(* Logix 5000 project; controller Good_Foods_96985_10252022_1208 vendor 1 type 14 code 151 rev 32.15; software revision 32.04; part 4 of 4 *)
(* tags used below, declared in another part *)
   Auto_Reset_Timer : TIMER;
   Auto_Reset_Timer2 : TIMER;
   bActive_Cleanout_Mode : BOOL;
   bAll_Doors_OK : BOOL;
   bAll_EStops_OK : BOOL;
   bAuto_Clear_Faults : BOOL;
   bAuto_Disable_Servos : BOOL;
   bAuto_Enable_Servos : BOOL;
   bAuto_Enable_VFDs : BOOL;
   bAuto_Reset_Latch : BOOL;
   bAuto_Reset_Servos : BOOL;
   bBatch_Cmplt : BOOL;
   bHMI_IND_Alarm_Active : BOOL;
   bHMI_IND_Servos_Enable : BOOL;
   bHMI_PB_Fault_Reset : BOOL;
   bHMI_PB_Jog_Infeed_Conveyors : BOOL;
   bHMI_PB_JogFwd_Left_Denester : BOOL;
   bHMI_PB_JogFwd_Right_Denester : BOOL;
   bHMI_PB_JogRev_Left_Denester : BOOL;
   bHMI_PB_JogRev_Right_Denester : BOOL;
   bHMI_PB_Left_Denester_Enabled : BOOL;
   bHMI_PB_Right_Denester_Enabled : BOOL;
   bLeft_System_Not_Running : BOOL;
   bLeftConvBacklog_OK : BOOL;
   bLeftDropBacklog_OK : BOOL;
   bLeftPrimeBacklog_OK : BOOL;
   bMachine_Startup_Delay : BOOL;
   bRight_System_Not_Running : BOOL;
   bRightConvBacklog_OK : BOOL;
   bRightDropBacklog_OK : BOOL;
   bRightPrimeBacklog_OK : BOOL;
   bSafety_OK : BOOL;
   bSystem_Active : BOOL;
   bSystem_Alarm_Active : BOOL;
   bSystem_Conveyor_Run_Perm : BOOL;
   bSystem_Needs_To_Be_Homed : BOOL;
   bSystem_VFDStop_CMPLT : BOOL;
   dAlarms : DINT[8];
   DI_Estop_Autoloader_Pressed : BOOL;
   DI_Estop_HMI_Pressed : BOOL;
   DI_Estop_NonOpSide_Pressed : BOOL;
   DI_PB_Autoloader_Start : BOOL;
   DI_PB_Hmi_Jog : BOOL;
   DI_PRX_Left_DropGate_EXT : BOOL;
   DI_PRX_Left_DropGate_RET : BOOL;
   DI_PRX_Left_Shuttle_RET : BOOL;
   DI_PRX_Right_DropGate_EXT : BOOL;
   DI_PRX_Right_DropGate_RET : BOOL;
   DI_PRX_Right_Shuttle_RET : BOOL;
   DI_PS_Air_Supply_OK : BOOL;
   DI_Safety_Relay_OK : BOOL;
   DI_SS_Left_NonOp_Door_Open : BOOL;
   DI_SS_Left_Op_Door_Open : BOOL;
   DI_SS_Right_NonOp_Door_Open : BOOL;
   DI_SS_Right_Op_Door_Open : BOOL;
   dLeft_Shuttle_Seq_CMD : DINT;
   dRight_Shuttle_Seq_CMD : DINT;
   intStatus_Message : INT;
   Left_Container_Jam_Timer : TIMER;
   Left_Denester : AXIS_CIP_DRIVE;
   Left_Rev_Count : INT;
   Master_Encoder : AXIS_CIP_DRIVE;
   ONS : DINT[16];
   rConv_Speed : REAL;
   rConv_Speed_Hz : DINT;
   rHMI_Infeed_Conv_Multiplier : REAL;
   rHMI_Machine_Speed : REAL;
   Right_Container_Jam_Timer : TIMER;
   Right_Denester : AXIS_CIP_DRIVE;
   Right_Rev_Count : INT;
   Timer_AirPressure : TIMER;
   tLeftDropGateContTimeOut : TIMER;
   tLeftDropGateExtTimeOut : TIMER;
   tLeftDropGateOpenTimeOut : TIMER;
   tLeftShuttleContPresTimeOut : TIMER;
   tloadconvpress : TIMER;
   tRightDropGateContTimeOut : TIMER;
   tRightDropGateExtTimeOut : TIMER;
   tRightDropGateOpenTimeOut : TIMER;
   tRightShuttleContPresTimeOut : TIMER;
(* MainProgram, continued *)

ROUTINE _30_VFDs   (* ladder *)
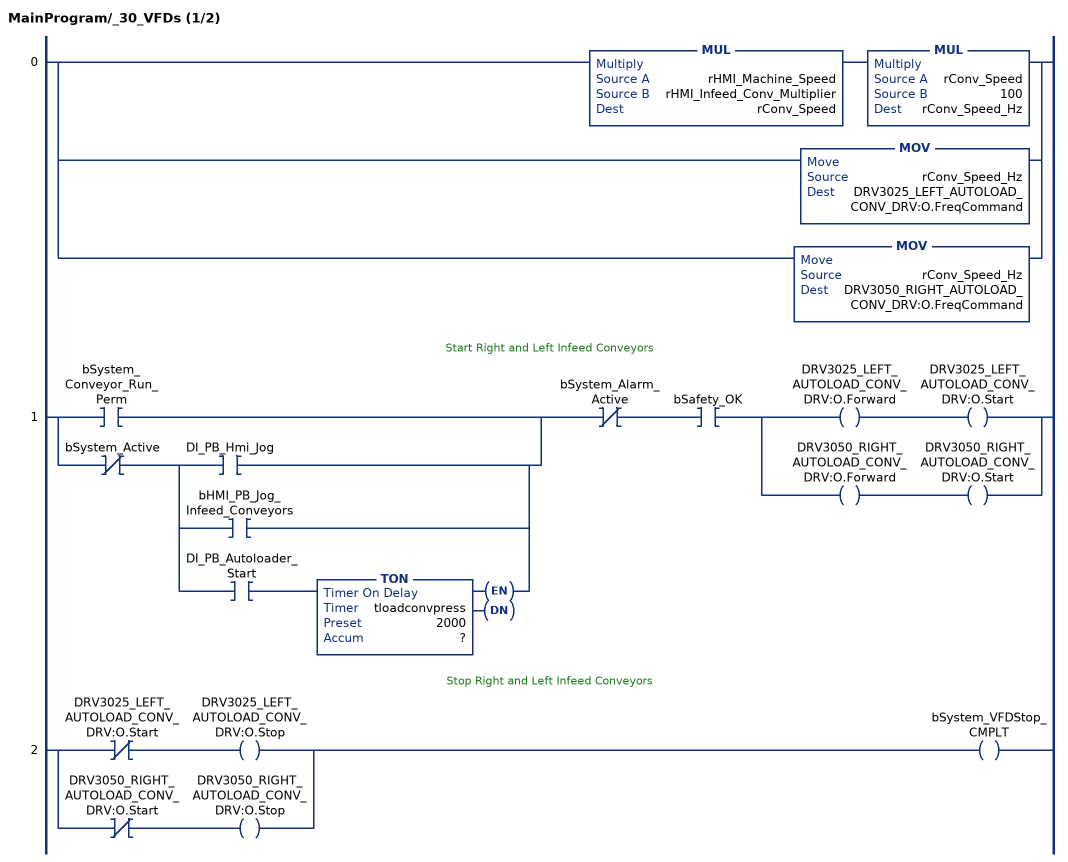
   0: [MUL(rHMI_Machine_Speed,rHMI_Infeed_Conv_Multiplier,rConv_Speed) MUL(rConv_Speed,100,rConv_Speed_Hz) ,MOV(rConv_Speed_Hz,DRV3025_LEFT_AUTOLOAD_CONV_DRV:O.FreqCommand) ,MOV(rConv_Speed_Hz,DRV3050_RIGHT_AUTOLOAD_CONV_DRV:O.FreqCommand) ];
   // Start Right and Left Infeed Conveyors
   1: [XIC(bSystem_Conveyor_Run_Perm) ,XIO(bSystem_Active) [XIC(DI_PB_Hmi_Jog) ,XIC(bHMI_PB_Jog_Infeed_Conveyors) ,XIC(DI_PB_Autoloader_Start) TON(tloadconvpress,?,?) ] ]XIO(bSystem_Alarm_Active)XIC(bSafety_OK)[OTE(DRV3025_LEFT_AUTOLOAD_CONV_DRV:O.Forward) OTE(DRV3025_LEFT_AUTOLOAD_CONV_DRV:O.Start) ,OTE(DRV3050_RIGHT_AUTOLOAD_CONV_DRV:O.Forward) OTE(DRV3050_RIGHT_AUTOLOAD_CONV_DRV:O.Start) ];
   // Stop Right and Left Infeed Conveyors
   2: [XIO(DRV3025_LEFT_AUTOLOAD_CONV_DRV:O.Start) OTE(DRV3025_LEFT_AUTOLOAD_CONV_DRV:O.Stop) ,XIO(DRV3050_RIGHT_AUTOLOAD_CONV_DRV:O.Start) OTE(DRV3050_RIGHT_AUTOLOAD_CONV_DRV:O.Stop) ]OTE(bSystem_VFDStop_CMPLT);
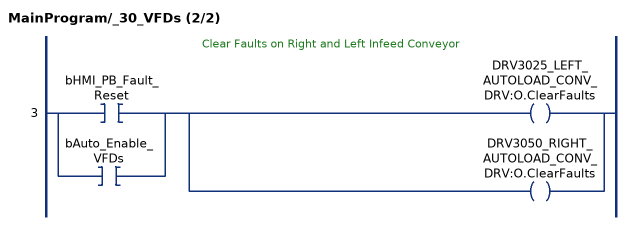
   // Clear Faults on Right and Left Infeed Conveyor
   3: [XIC(bHMI_PB_Fault_Reset) ,XIC(bAuto_Enable_VFDs) ][OTE(DRV3025_LEFT_AUTOLOAD_CONV_DRV:O.ClearFaults) ,OTE(DRV3050_RIGHT_AUTOLOAD_CONV_DRV:O.ClearFaults) ];
END_ROUTINE

ROUTINE _90_Status_Messages   (* ladder *)
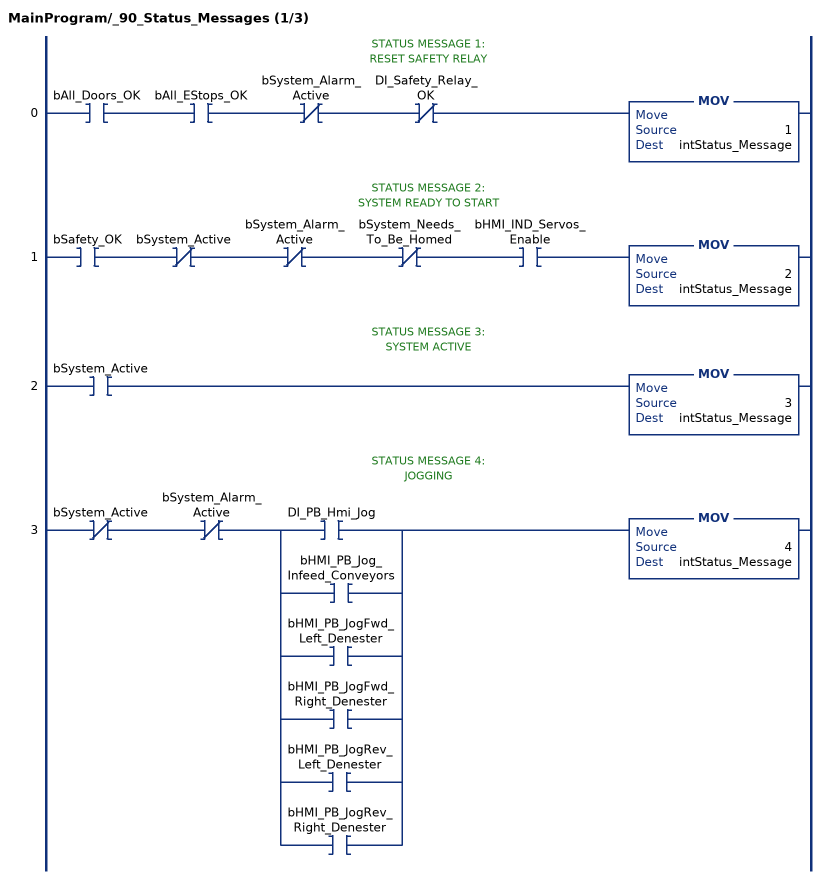
   // STATUS MESSAGE 1:
   // RESET SAFETY RELAY
   0: XIC(bAll_Doors_OK)XIC(bAll_EStops_OK)XIO(bSystem_Alarm_Active)XIO(DI_Safety_Relay_OK)MOV(1,intStatus_Message);
   // STATUS MESSAGE 2:
   // SYSTEM READY TO START
   1: XIC(bSafety_OK)XIO(bSystem_Active)XIO(bSystem_Alarm_Active)XIO(bSystem_Needs_To_Be_Homed)XIC(bHMI_IND_Servos_Enable)MOV(2,intStatus_Message);
   // STATUS MESSAGE 3:
   // SYSTEM ACTIVE
   2: XIC(bSystem_Active)MOV(3,intStatus_Message);
   // STATUS MESSAGE 4:
   // JOGGING
   3: XIO(bSystem_Active)XIO(bSystem_Alarm_Active)[XIC(DI_PB_Hmi_Jog) ,XIC(bHMI_PB_Jog_Infeed_Conveyors) ,XIC(bHMI_PB_JogFwd_Left_Denester) ,XIC(bHMI_PB_JogFwd_Right_Denester) ,XIC(bHMI_PB_JogRev_Left_Denester) ,XIC(bHMI_PB_JogRev_Right_Denester) ]MOV(4,intStatus_Message);
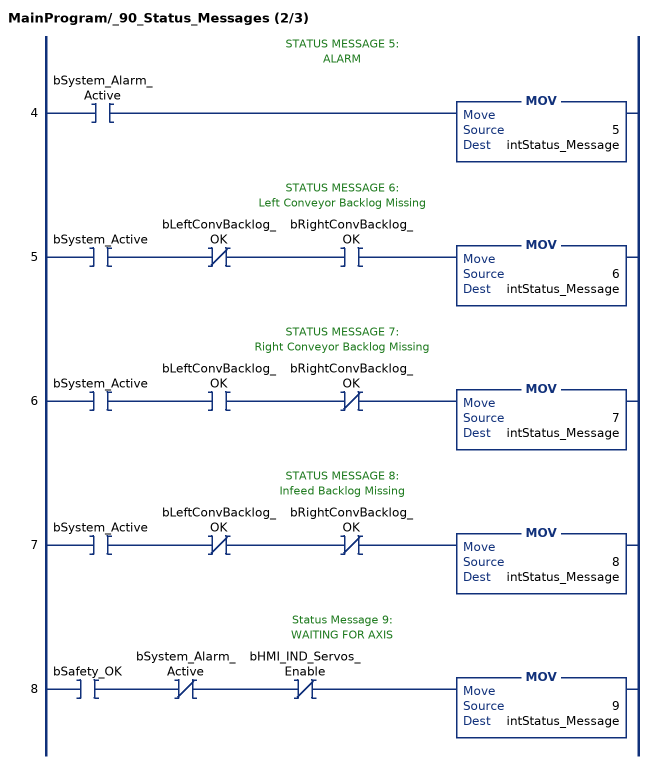
   // STATUS MESSAGE 5:
   // ALARM
   4: XIC(bSystem_Alarm_Active)MOV(5,intStatus_Message);
   // STATUS MESSAGE 6:
   // Left Conveyor Backlog Missing
   5: XIC(bSystem_Active)XIO(bLeftConvBacklog_OK)XIC(bRightConvBacklog_OK)MOV(6,intStatus_Message);
   // STATUS MESSAGE 7:
   // Right Conveyor Backlog Missing
   6: XIC(bSystem_Active)XIC(bLeftConvBacklog_OK)XIO(bRightConvBacklog_OK)MOV(7,intStatus_Message);
   // STATUS MESSAGE 8:
   // Infeed Backlog Missing
   7: XIC(bSystem_Active)XIO(bLeftConvBacklog_OK)XIO(bRightConvBacklog_OK)MOV(8,intStatus_Message);
   // Status Message 9:
   // WAITING FOR AXIS
   8: XIC(bSafety_OK)XIO(bSystem_Alarm_Active)XIO(bHMI_IND_Servos_Enable)MOV(9,intStatus_Message);
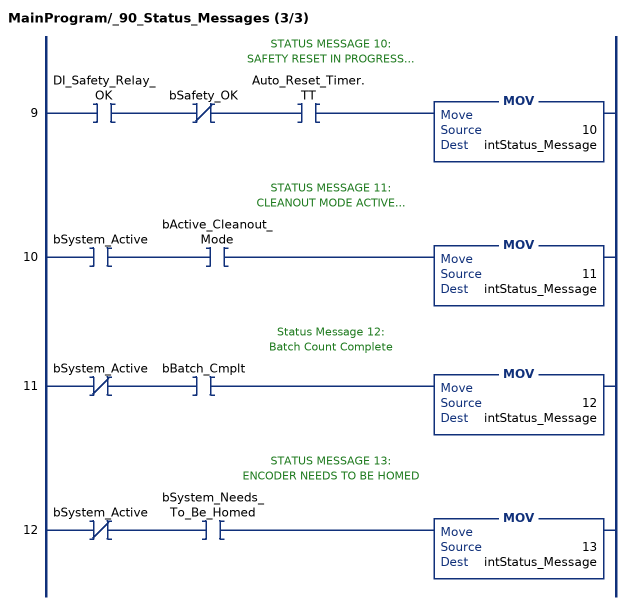
   // STATUS MESSAGE 10:
   // SAFETY RESET IN PROGRESS...
   9: XIC(DI_Safety_Relay_OK)XIO(bSafety_OK)XIC(Auto_Reset_Timer.TT)MOV(10,intStatus_Message);
   // STATUS MESSAGE 11:
   // CLEANOUT MODE ACTIVE...
   10: XIC(bSystem_Active)XIC(bActive_Cleanout_Mode)MOV(11,intStatus_Message);
   // Status Message 12:
   // Batch Count Complete
   11: XIO(bSystem_Active)XIC(bBatch_Cmplt)MOV(12,intStatus_Message);
   // STATUS MESSAGE 13:
   // ENCODER NEEDS TO BE HOMED
   12: XIO(bSystem_Active)XIC(bSystem_Needs_To_Be_Homed)MOV(13,intStatus_Message);
END_ROUTINE

ROUTINE _99_Alarms   (* ladder *)
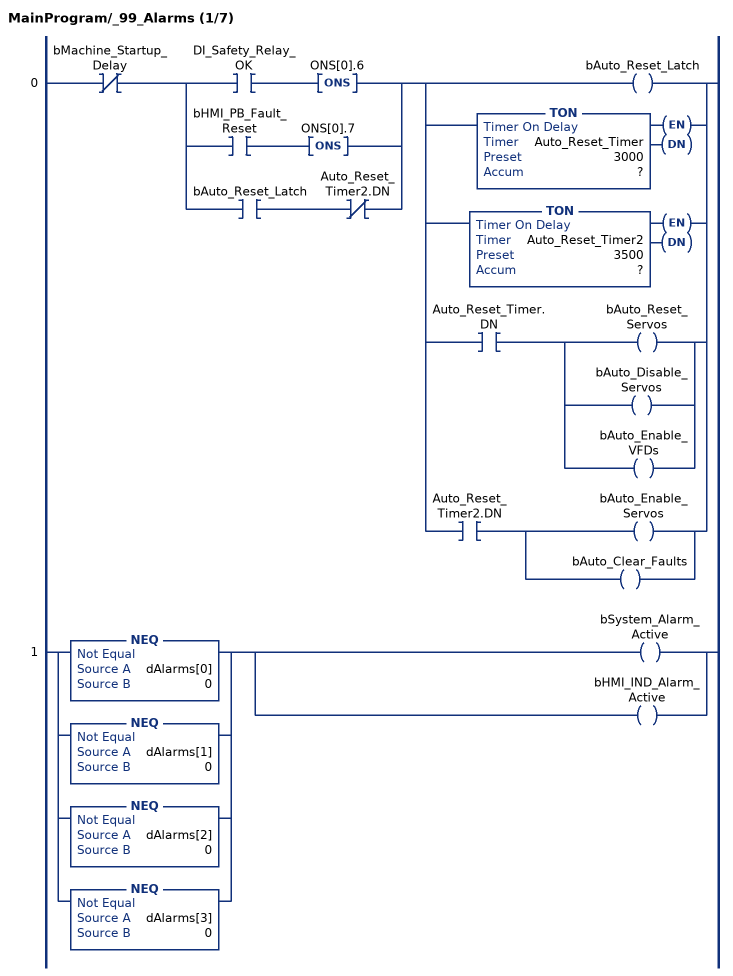
   0: XIO(bMachine_Startup_Delay)[XIC(DI_Safety_Relay_OK) ONS(ONS[0].6) ,XIC(bHMI_PB_Fault_Reset) ONS(ONS[0].7) ,XIC(bAuto_Reset_Latch) XIO(Auto_Reset_Timer2.DN) ][OTE(bAuto_Reset_Latch) ,TON(Auto_Reset_Timer,?,?) ,TON(Auto_Reset_Timer2,?,?) ,XIC(Auto_Reset_Timer.DN) [OTE(bAuto_Reset_Servos) ,OTE(bAuto_Disable_Servos) ,OTE(bAuto_Enable_VFDs) ] ,XIC(Auto_Reset_Timer2.DN) [OTE(bAuto_Enable_Servos) ,OTE(bAuto_Clear_Faults) ] ];
   1: [NEQ(dAlarms[0],0) ,NEQ(dAlarms[1],0) ,NEQ(dAlarms[2],0) ,NEQ(dAlarms[3],0) ][OTE(bSystem_Alarm_Active) ,OTE(bHMI_IND_Alarm_Active) ];
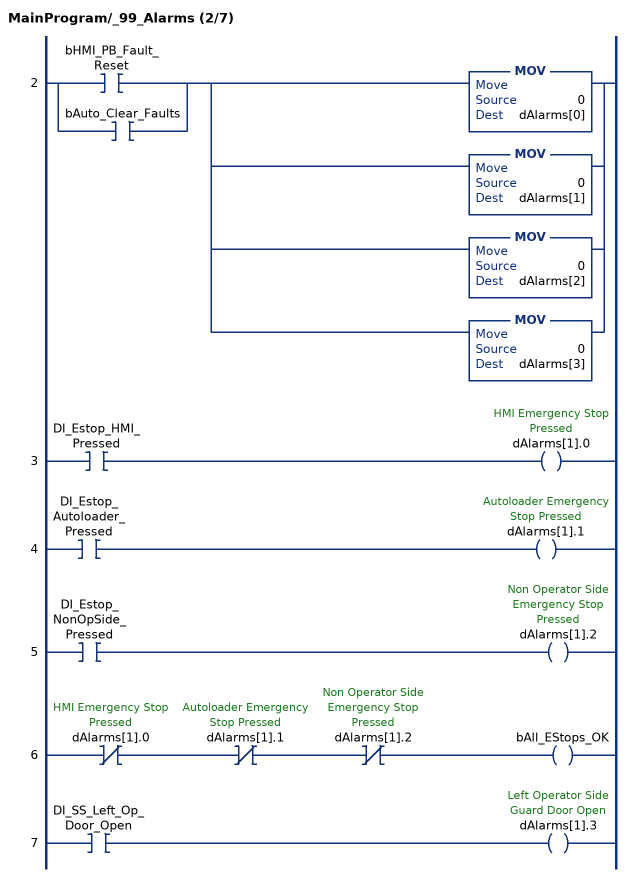
   2: [XIC(bHMI_PB_Fault_Reset) ,XIC(bAuto_Clear_Faults) ][MOV(0,dAlarms[0]) ,MOV(0,dAlarms[1]) ,MOV(0,dAlarms[2]) ,MOV(0,dAlarms[3]) ];
   3: XIC(DI_Estop_HMI_Pressed)OTE(dAlarms[1].0);
   4: XIC(DI_Estop_Autoloader_Pressed)OTE(dAlarms[1].1);
   5: XIC(DI_Estop_NonOpSide_Pressed)OTE(dAlarms[1].2);
   6: XIO(dAlarms[1].0)XIO(dAlarms[1].1)XIO(dAlarms[1].2)OTE(bAll_EStops_OK);
   7: XIC(DI_SS_Left_Op_Door_Open)OTE(dAlarms[1].3);
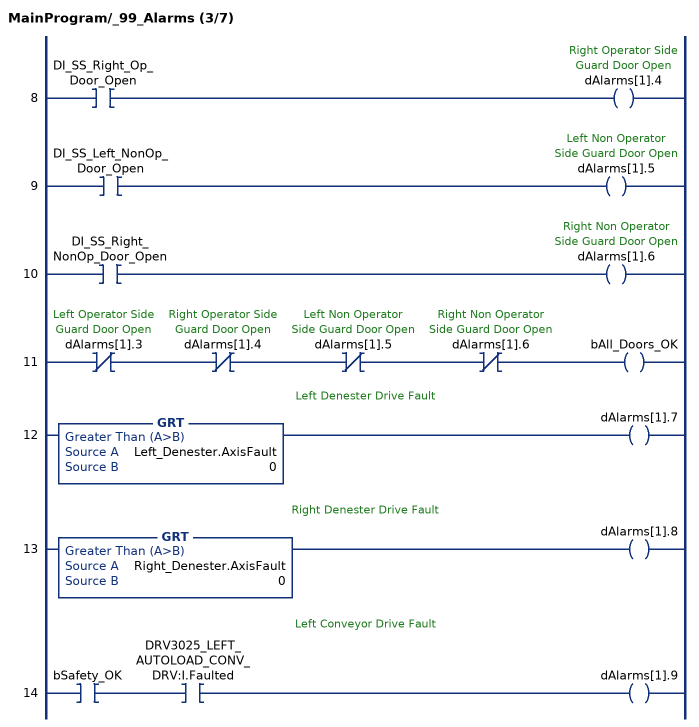
   8: XIC(DI_SS_Right_Op_Door_Open)OTE(dAlarms[1].4);
   9: XIC(DI_SS_Left_NonOp_Door_Open)OTE(dAlarms[1].5);
   10: XIC(DI_SS_Right_NonOp_Door_Open)OTE(dAlarms[1].6);
   11: XIO(dAlarms[1].3)XIO(dAlarms[1].4)XIO(dAlarms[1].5)XIO(dAlarms[1].6)OTE(bAll_Doors_OK);
   // Left Denester Drive Fault
   12: GRT(Left_Denester.AxisFault,0)OTE(dAlarms[1].7);
   // Right Denester Drive Fault
   13: GRT(Right_Denester.AxisFault,0)OTE(dAlarms[1].8);
   // Left Conveyor Drive Fault
   14: XIC(bSafety_OK)XIC(DRV3025_LEFT_AUTOLOAD_CONV_DRV:I.Faulted)OTE(dAlarms[1].9);
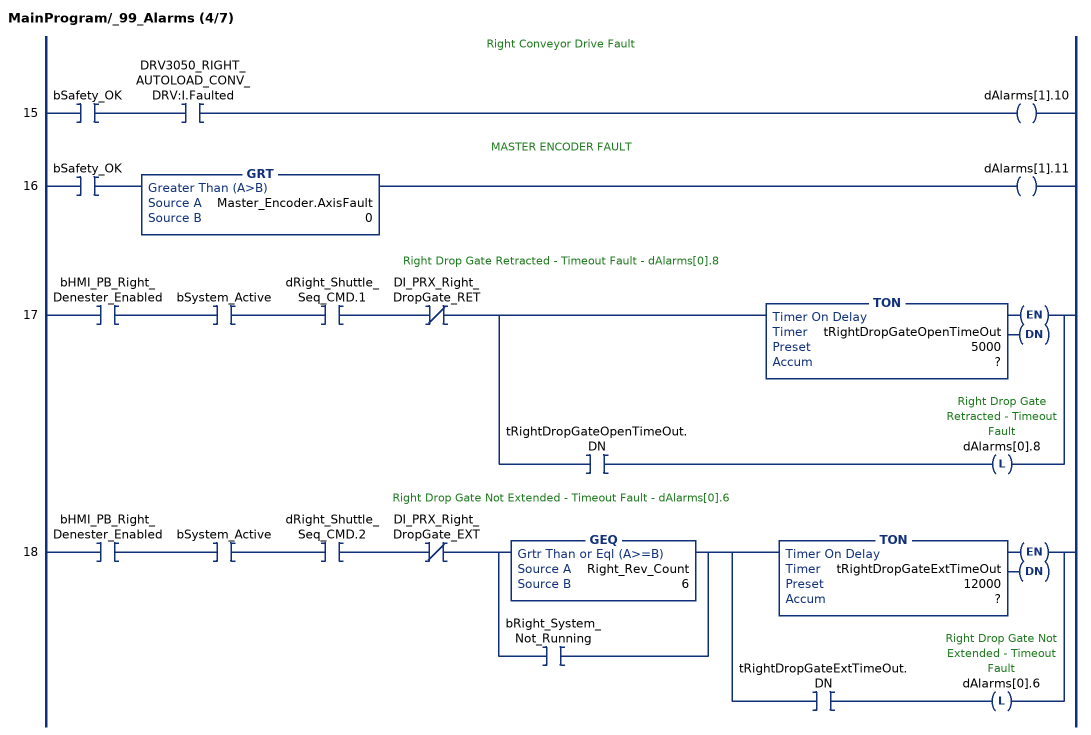
   // Right Conveyor Drive Fault
   15: XIC(bSafety_OK)XIC(DRV3050_RIGHT_AUTOLOAD_CONV_DRV:I.Faulted)OTE(dAlarms[1].10);
   // MASTER ENCODER FAULT
   16: XIC(bSafety_OK)GRT(Master_Encoder.AxisFault,0)OTE(dAlarms[1].11);
   // Right Drop Gate Retracted - Timeout Fault - dAlarms[0].8
   17: XIC(bHMI_PB_Right_Denester_Enabled)XIC(bSystem_Active)XIC(dRight_Shuttle_Seq_CMD.1)XIO(DI_PRX_Right_DropGate_RET)[TON(tRightDropGateOpenTimeOut,?,?) ,XIC(tRightDropGateOpenTimeOut.DN) OTL(dAlarms[0].8) ];
   // Right Drop Gate Not Extended - Timeout Fault - dAlarms[0].6
   18: XIC(bHMI_PB_Right_Denester_Enabled)XIC(bSystem_Active)XIC(dRight_Shuttle_Seq_CMD.2)XIO(DI_PRX_Right_DropGate_EXT)[GEQ(Right_Rev_Count,6) ,XIC(bRight_System_Not_Running) ][TON(tRightDropGateExtTimeOut,?,?) ,XIC(tRightDropGateExtTimeOut.DN) OTL(dAlarms[0].6) ];
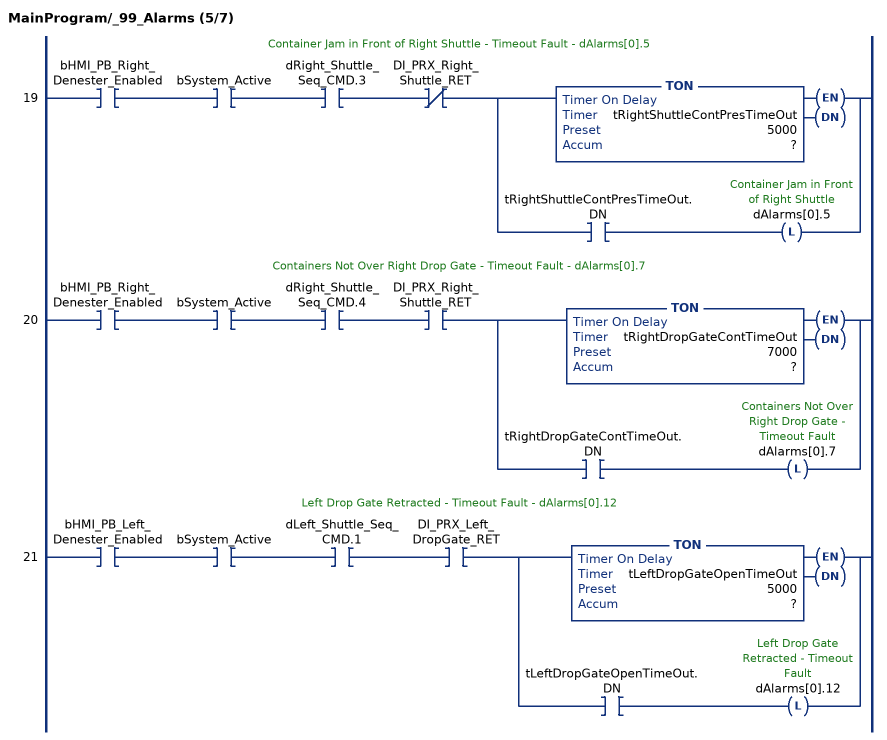
   // Container Jam in Front of Right Shuttle - Timeout Fault - dAlarms[0].5
   19: XIC(bHMI_PB_Right_Denester_Enabled)XIC(bSystem_Active)XIC(dRight_Shuttle_Seq_CMD.3)XIO(DI_PRX_Right_Shuttle_RET)[TON(tRightShuttleContPresTimeOut,?,?) ,XIC(tRightShuttleContPresTimeOut.DN) OTL(dAlarms[0].5) ];
   // Containers Not Over Right Drop Gate - Timeout Fault - dAlarms[0].7
   20: XIC(bHMI_PB_Right_Denester_Enabled)XIC(bSystem_Active)XIC(dRight_Shuttle_Seq_CMD.4)XIC(DI_PRX_Right_Shuttle_RET)[TON(tRightDropGateContTimeOut,?,?) ,XIC(tRightDropGateContTimeOut.DN) OTL(dAlarms[0].7) ];
   // Left Drop Gate Retracted - Timeout Fault - dAlarms[0].12
   21: XIC(bHMI_PB_Left_Denester_Enabled)XIC(bSystem_Active)XIC(dLeft_Shuttle_Seq_CMD.1)XIC(DI_PRX_Left_DropGate_RET)[TON(tLeftDropGateOpenTimeOut,?,?) ,XIC(tLeftDropGateOpenTimeOut.DN) OTL(dAlarms[0].12) ];
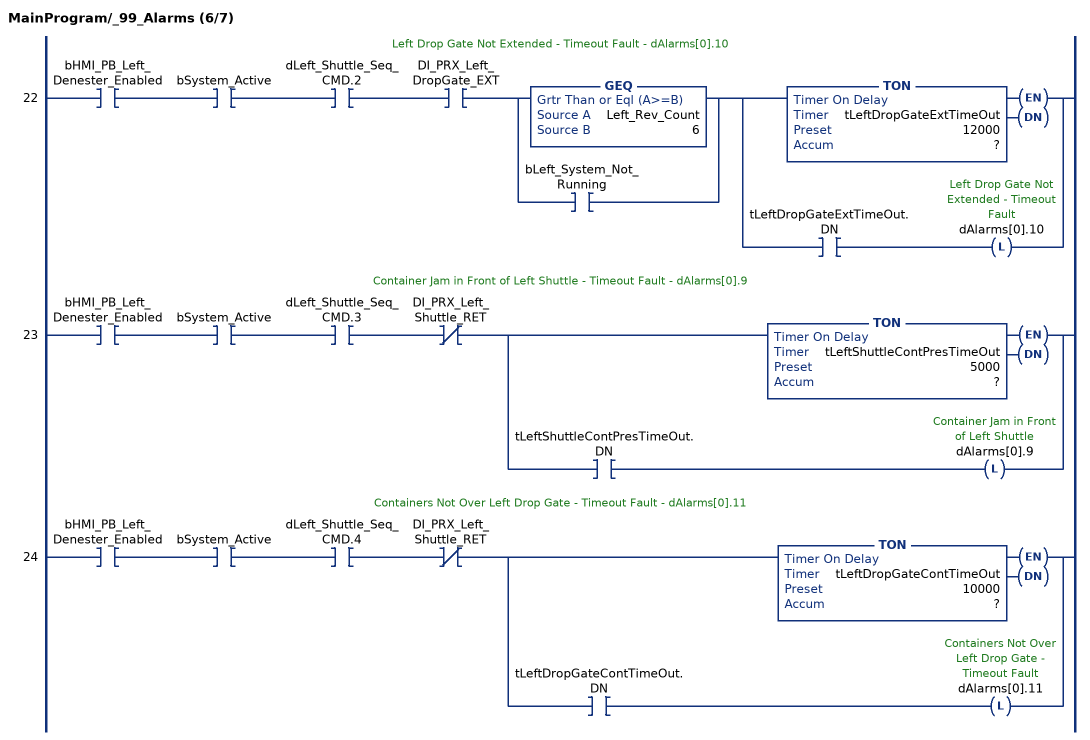
   // Left Drop Gate Not Extended - Timeout Fault - dAlarms[0].10
   22: XIC(bHMI_PB_Left_Denester_Enabled)XIC(bSystem_Active)XIC(dLeft_Shuttle_Seq_CMD.2)XIC(DI_PRX_Left_DropGate_EXT)[GEQ(Left_Rev_Count,6) ,XIC(bLeft_System_Not_Running) ][TON(tLeftDropGateExtTimeOut,?,?) ,XIC(tLeftDropGateExtTimeOut.DN) OTL(dAlarms[0].10) ];
   // Container Jam in Front of Left Shuttle - Timeout Fault - dAlarms[0].9
   23: XIC(bHMI_PB_Left_Denester_Enabled)XIC(bSystem_Active)XIC(dLeft_Shuttle_Seq_CMD.3)XIO(DI_PRX_Left_Shuttle_RET)[TON(tLeftShuttleContPresTimeOut,?,?) ,XIC(tLeftShuttleContPresTimeOut.DN) OTL(dAlarms[0].9) ];
   // Containers Not Over Left Drop Gate - Timeout Fault - dAlarms[0].11
   24: XIC(bHMI_PB_Left_Denester_Enabled)XIC(bSystem_Active)XIC(dLeft_Shuttle_Seq_CMD.4)XIO(DI_PRX_Left_Shuttle_RET)[TON(tLeftDropGateContTimeOut,?,?) ,XIC(tLeftDropGateContTimeOut.DN) OTL(dAlarms[0].11) ];
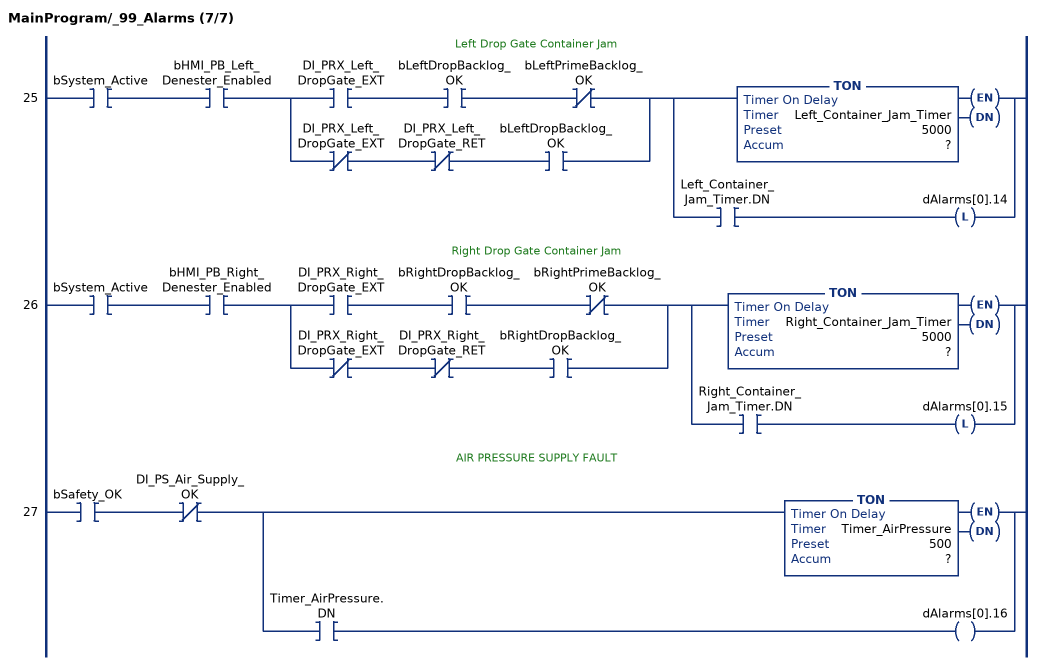
   // Left Drop Gate Container Jam
   25: XIC(bSystem_Active)XIC(bHMI_PB_Left_Denester_Enabled)[XIC(DI_PRX_Left_DropGate_EXT) XIC(bLeftDropBacklog_OK) XIO(bLeftPrimeBacklog_OK) ,XIO(DI_PRX_Left_DropGate_EXT) XIO(DI_PRX_Left_DropGate_RET) XIC(bLeftDropBacklog_OK) ][TON(Left_Container_Jam_Timer,?,?) ,XIC(Left_Container_Jam_Timer.DN) OTL(dAlarms[0].14) ];
   // Right Drop Gate Container Jam
   26: XIC(bSystem_Active)XIC(bHMI_PB_Right_Denester_Enabled)[XIC(DI_PRX_Right_DropGate_EXT) XIC(bRightDropBacklog_OK) XIO(bRightPrimeBacklog_OK) ,XIO(DI_PRX_Right_DropGate_EXT) XIO(DI_PRX_Right_DropGate_RET) XIC(bRightDropBacklog_OK) ][TON(Right_Container_Jam_Timer,?,?) ,XIC(Right_Container_Jam_Timer.DN) OTL(dAlarms[0].15) ];
   // AIR PRESSURE SUPPLY FAULT
   27: XIC(bSafety_OK)XIO(DI_PS_Air_Supply_OK)[TON(Timer_AirPressure,?,?) ,XIC(Timer_AirPressure.DN) OTE(dAlarms[0].16) ];
END_ROUTINE
END_PROGRAM
